// TIA Portal V16 export
// export: Created 2023-08-28T09:37:38.4418764Z, ExportSetting WithDefaults, DisplayName Totally Integrated Automation Portal, DisplayVersion V16 Update 6, DisplayName TIA Portal Version Control Interface, DisplayVersion V16 Update 2, DisplayName TIA Portal Openness, DisplayVersion V16 Update 6, DisplayName STEP 7 Professional, DisplayVersion V16 Update 6, DisplayName STEP 7 Safety, DisplayVersion V16, DisplayName WinCC Advanced, DisplayVersion V16 Update 6
FUNCTION "08_C_Detection_Changes_Data_Word" : Void   // FC62, LAD
{ S7_Optimized_Access := 'TRUE' }
AUTHOR : rtecmer
VERSION : 0.1
// stored: AutoNumber false, IsIECCheckEnabled false, SetENOAutomatically false, UDAEnableTagReadback false
   VAR_IN_OUT
      "dbHold_Sending_TCP.Sending_Hold" : Int;   // Zmienna zadająca i porównywana
      dbHoldRegSlave_to_MT101 : Int;   // Zmienna w db do której porównujemy
      memRisingTriger_Data_ : Bool;   // bit pamięć zmiany
      "dbHold_RRG.Sending" : Int;   // zmienna docelowa w db do wysłania
   END_VAR
   VAR_TEMP   // added for the SCL form of the ladder/FBD networks
      _w1 : Bool;
      _w2 : Bool;
   END_VAR
BEGIN

REGION Network 1: set_poziom_napełniania
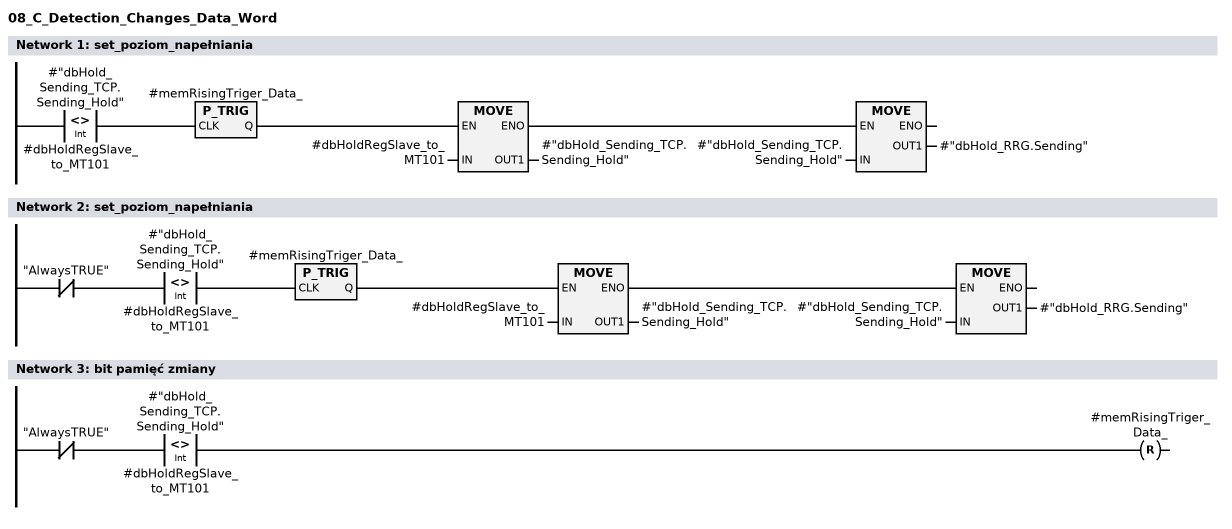
   RUNG wire#powerrail
      { S7_Templates := "SrcType := Int" } NE_Contact(in1 := #"dbHold_Sending_TCP.Sending_Hold", in2 := #dbHoldRegSlave_to_MT101)
      P_Trig( #memRisingTriger_Data_ )
      Move(in := #dbHoldRegSlave_to_MT101, out1 => #"dbHold_Sending_TCP.Sending_Hold")
      Move(in := #"dbHold_Sending_TCP.Sending_Hold", out1 => #"dbHold_RRG.Sending")
   END_RUNG
   // the same network as SCL:
   #_w1 := #"dbHold_Sending_TCP.Sending_Hold" <> #dbHoldRegSlave_to_MT101;
   #_w2 := #_w1 AND NOT #memRisingTriger_Data_;   // rising edge
   #memRisingTriger_Data_ := #_w1;
   IF #_w2 THEN
       #"dbHold_Sending_TCP.Sending_Hold" := #dbHoldRegSlave_to_MT101;
       #"dbHold_RRG.Sending" := #"dbHold_Sending_TCP.Sending_Hold";
   END_IF;
END_REGION

REGION Network 2: set_poziom_napełniania
   RUNG wire#powerrail
      I_Contact( "AlwaysTRUE" )
      { S7_Templates := "SrcType := Int" } NE_Contact(in1 := #"dbHold_Sending_TCP.Sending_Hold", in2 := #dbHoldRegSlave_to_MT101)
      P_Trig( #memRisingTriger_Data_ )
      Move(in := #dbHoldRegSlave_to_MT101, out1 => #"dbHold_Sending_TCP.Sending_Hold")
      Move(in := #"dbHold_Sending_TCP.Sending_Hold", out1 => #"dbHold_RRG.Sending")
   END_RUNG
   // the same network as SCL:
   #_w1 := NOT "AlwaysTRUE" AND (#"dbHold_Sending_TCP.Sending_Hold" <> #dbHoldRegSlave_to_MT101);
   #_w2 := #_w1 AND NOT #memRisingTriger_Data_;   // rising edge
   #memRisingTriger_Data_ := #_w1;
   IF #_w2 THEN
       #"dbHold_Sending_TCP.Sending_Hold" := #dbHoldRegSlave_to_MT101;
       #"dbHold_RRG.Sending" := #"dbHold_Sending_TCP.Sending_Hold";
   END_IF;
END_REGION

REGION Network 3: bit pamięć zmiany
   RUNG wire#powerrail
      I_Contact( "AlwaysTRUE" )
      { S7_Templates := "SrcType := Int" } NE_Contact(in1 := #"dbHold_Sending_TCP.Sending_Hold", in2 := #dbHoldRegSlave_to_MT101)
      R_Coil( #memRisingTriger_Data_ )
   END_RUNG
   // the same network as SCL:
   IF NOT "AlwaysTRUE" AND (#"dbHold_Sending_TCP.Sending_Hold" <> #dbHoldRegSlave_to_MT101) THEN
       #memRisingTriger_Data_ := FALSE;
   END_IF;
END_REGION
END_FUNCTION
